(* Logix 5000 project; controller Capstone_PLC_1 1769-L16ER-BB1B rev 38.11; software revision 38.00; part 2 of 2 *)
(* tags used below, declared in another part *)
   Cmd_Conv : ALIAS FOR Point_IO:3:O.0;   // Logically commands conveyor output
   Cmd_Eject_1 : ALIAS FOR Point_IO:3:O.1;   // Logically commands ejection nozzle 1 output
   Cmd_Eject_2 : ALIAS FOR Point_IO:3:O.2;   // Logically commands ejection nozzle 2 output
   Cmd_Eject_3 : ALIAS FOR Point_IO:3:O.3;   // Logically commands ejection nozzle 3 output
   Color_Code : DINT;   // Detected color code
   ColorValid : BOOL;   // Validates color reading
   Con_0 : DINT;   // Constant 0
   Con_1 : DINT;   // Constant 1
   Con_2 : DINT;   // Constant 2
   Con_4 : DINT;   // Constant 4
   Count_1 : DINT;   // Bin 1 counter
   Count_2 : DINT;   // Bin 2 counter
   Count_3 : DINT;   // Bin 3 counter
   Count_4 : DINT;   // Bin 4 counter
   Dest_Bin : DINT;   // Stores destination bin after a cube is identified
   DONE : DINT;   // State, cube sorted, triggers check, if cubes left to be sorted State returns to PICK, if not State returns to IDLE
   IDLE : DINT;   // State, system is initialized but no tray is present or tray present with no cubes
   Ind_Tray_1 : ALIAS FOR Point_IO:1:I.1;   // Induction sensor 1: Tray identification
   Ind_Tray_2 : ALIAS FOR Point_IO:1:I.2;   // Induction sensor 2: Tray identification
   Ind_Tray_3 : ALIAS FOR Point_IO:1:I.3;   // Induction sensor 3: Tray identification
   Lim_Tray_Pres : ALIAS FOR Point_IO:1:I.0;   // Limit switch: Tray presence
   OS_TrayID_1 : BOOL;   // Protects from induction sensor reading multipletimes
   OS_TrayID_2 : BOOL;   // Protects from induction sensor reading multipletimes
   OS_TrayID_3 : BOOL;   // Protects from induction sensor reading multipletimes
   Output_Enable : BOOL;   // Enables outputs if robot initialized, system in run mode, and no faults or estop
   PICK : DINT;   // State, robot picking
   Pick_Done : BOOL;   // Triggers when SPEL pick is completed
   Pick_Index : DINT;   // Tracks cubes on tray for picking
   READY : DINT;   // State, Tray and cubes present
   SCADA_Color : DINT;   // SCADA tag shows identified color
   SCADA_Count_1 : DINT;   // SCADA tag shows counter for bin 1
   SCADA_Count_2 : DINT;   // SCADA tag shows counter for bin 2
   SCADA_Count_3 : DINT;   // SCADA tag shows counter for bin 3
   SCADA_Count_4 : DINT;   // SCADA tag shows counter for bin 4
   SCADA_Dest : DINT;   // SCADA tag shows destination bin
   SCADA_State : DINT;   // SCADA tag shows current system state
   SCADA_TrayID : DINT;   // SCADA tag shows Tray ID
   State : DINT;   // Tracks system state for control flow
   Sys_Rdy : BOOL;   // System staged and safe for production
   Sys_Run : BOOL;   // Production active
   Thr_Cubes_1 : ALIAS FOR Point_IO:1:I.4;   // Through beam sensor: identifies cube presence in tray row 1
   Thr_Cubes_2 : ALIAS FOR Point_IO:1:I.5;   // Through beam sensor: identifies cube presence in tray row 2
   Tray_Full : BOOL;   // Energizes if both through beam sensors are triggered for cube presence
   TrayID : DINT;   // Calculated tray ID from induction sensors
   TrayIdentified : BOOL;   // Tracks if a tray is identified
(* MainProgram, continued *)

ROUTINE SCADA_Mapping   (* ladder *)
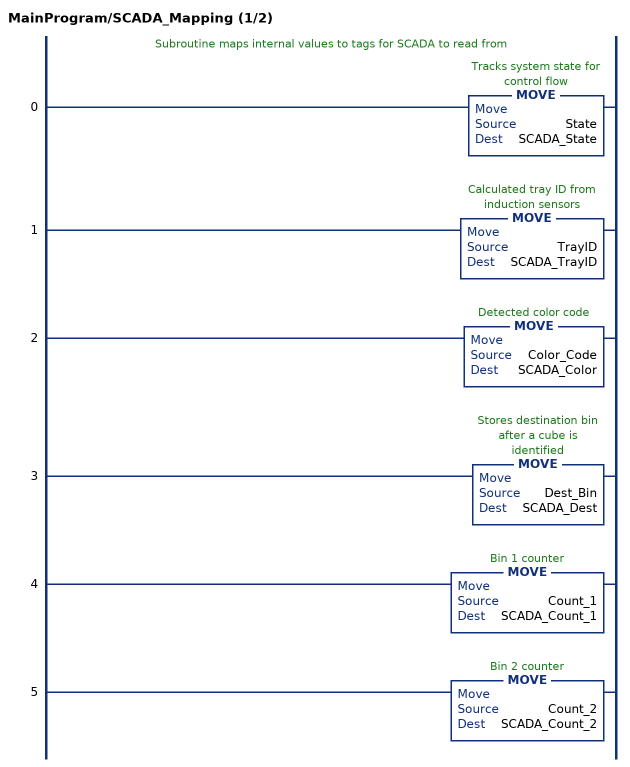
   // Subroutine maps internal values to tags for SCADA to read from
   0: MOVE(State,SCADA_State);
   1: MOVE(TrayID,SCADA_TrayID);
   2: MOVE(Color_Code,SCADA_Color);
   3: MOVE(Dest_Bin,SCADA_Dest);
   4: MOVE(Count_1,SCADA_Count_1);
   5: MOVE(Count_2,SCADA_Count_2);
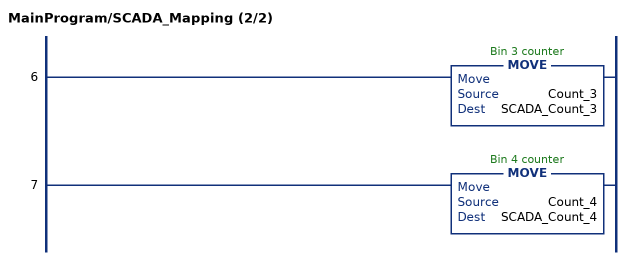
   6: MOVE(Count_3,SCADA_Count_3);
   7: MOVE(Count_4,SCADA_Count_4);
END_ROUTINE

ROUTINE System_Reset   (* ladder *)
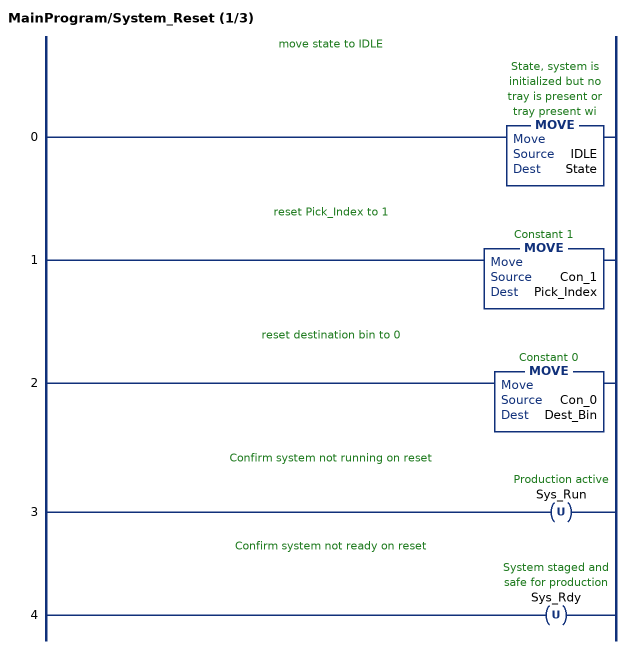
   // move state to IDLE
   0: MOVE(IDLE,State);
   // reset Pick_Index to 1
   1: MOVE(Con_1,Pick_Index);
   // reset destination bin to 0
   2: MOVE(Con_0,Dest_Bin);
   // Confirm system not running on reset
   3: OTU(Sys_Run);
   // Confirm system not ready on reset
   4: OTU(Sys_Rdy);
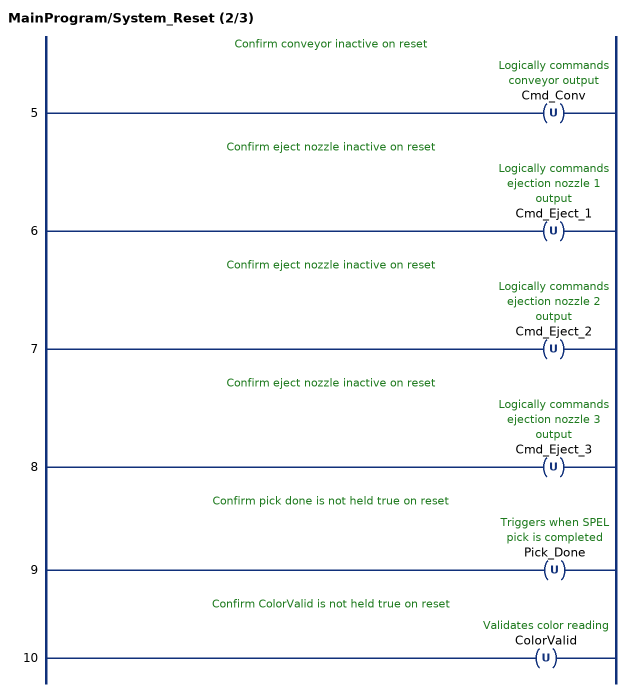
   // Confirm conveyor inactive on reset
   5: OTU(Cmd_Conv);
   // Confirm eject nozzle inactive on reset
   6: OTU(Cmd_Eject_1);
   // Confirm eject nozzle inactive on reset
   7: OTU(Cmd_Eject_2);
   // Confirm eject nozzle inactive on reset
   8: OTU(Cmd_Eject_3);
   // Confirm pick done is not held true on reset
   9: OTU(Pick_Done);
   // Confirm ColorValid is not held true on reset
   10: OTU(ColorValid);
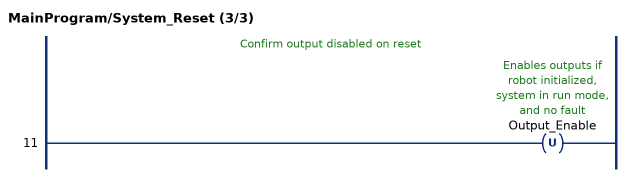
   // Confirm output disabled on reset
   11: OTU(Output_Enable);
END_ROUTINE

ROUTINE Tray_Identify   (* ladder *)
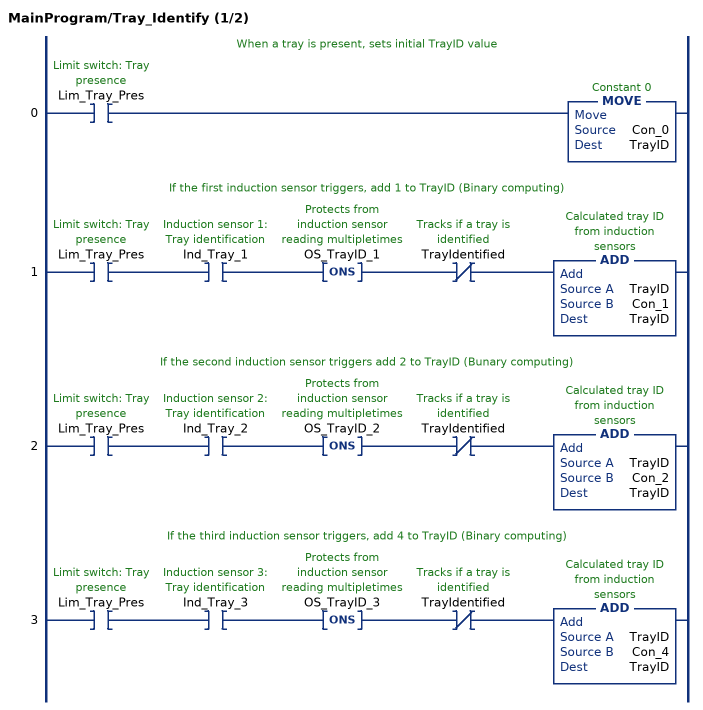
   // When a tray is present, sets initial TrayID value
   0: XIC(Lim_Tray_Pres)MOVE(Con_0,TrayID);
   // If the first induction sensor triggers, add 1 to TrayID (Binary computing)
   1: XIC(Lim_Tray_Pres)XIC(Ind_Tray_1)ONS(OS_TrayID_1)XIO(TrayIdentified)ADD(TrayID,Con_1,TrayID);
   // If the second induction sensor triggers add 2 to TrayID (Bunary computing)
   2: XIC(Lim_Tray_Pres)XIC(Ind_Tray_2)ONS(OS_TrayID_2)XIO(TrayIdentified)ADD(TrayID,Con_2,TrayID);
   // If the third induction sensor triggers, add 4 to TrayID (Binary computing)
   3: XIC(Lim_Tray_Pres)XIC(Ind_Tray_3)ONS(OS_TrayID_3)XIO(TrayIdentified)ADD(TrayID,Con_4,TrayID);
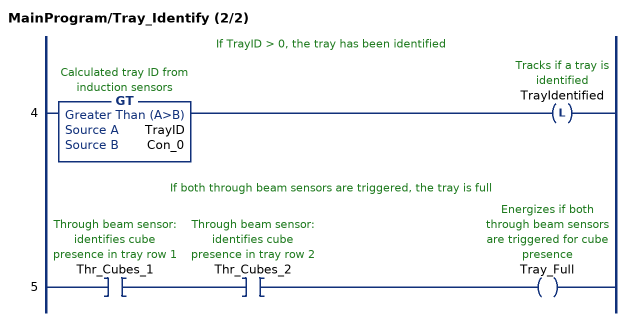
   // If TrayID > 0, the tray has been identified
   4: GT(TrayID,Con_0)OTL(TrayIdentified);
   // If both through beam sensors are triggered, the tray is full
   5: XIC(Thr_Cubes_1)XIC(Thr_Cubes_2)OTE(Tray_Full);
END_ROUTINE
END_PROGRAM

PROGRAM SecondaryProgram
END_PROGRAM
